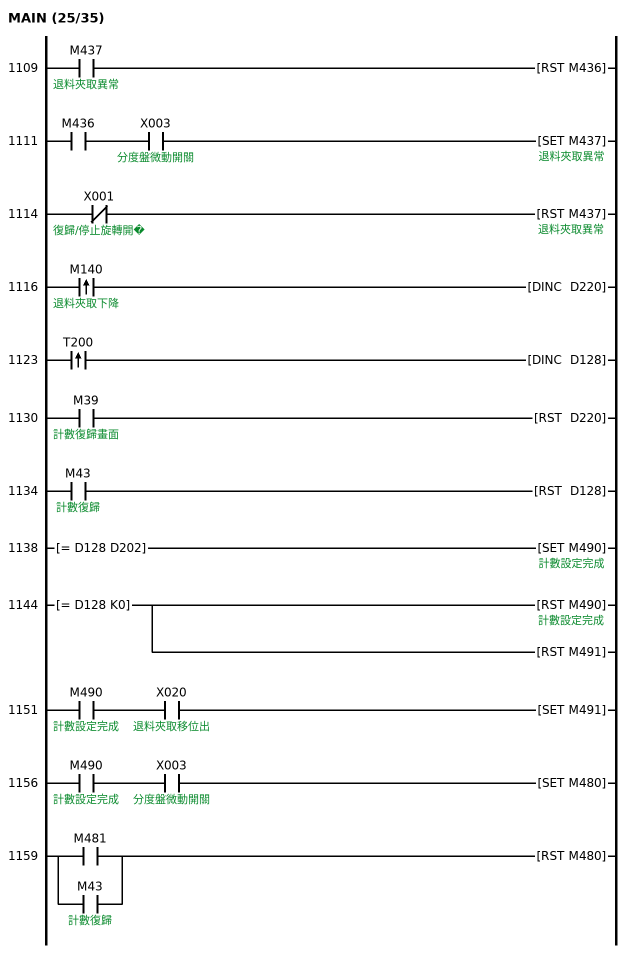
[picture p24: ladder of MAIN, rungs at steps 1109 to 1159]
1109  LD      M437  ; 退料夾取異常
      RST     M436
1111  LD      M436
      AND     X003  ; 分度盤微動開關
      SET     M437  ; 退料夾取異常
1114  LDI     X001  ; 復歸/停止旋轉開�
      RST     M437  ; 退料夾取異常
1116  LDP     M140  ; 退料夾取下降
      DINC    D220
1123  LDP     T200
      DINC    D128
1130  LD      M39  ; 計數復歸畫面
      RST     D220
1134  LD      M43  ; 計數復歸
      RST     D128
1138  LD=     D128 D202
      SET     M490  ; 計數設定完成
1144  LD=     D128 K0
      RST     M490  ; 計數設定完成
      RST     M491
1151  LD      M490  ; 計數設定完成
      AND     X020  ; 退料夾取移位出
      SET     M491
1156  LD      M490  ; 計數設定完成
      AND     X003  ; 分度盤微動開關
      SET     M480
1159  LD      M481
      OR      M43  ; 計數復歸
      RST     M480
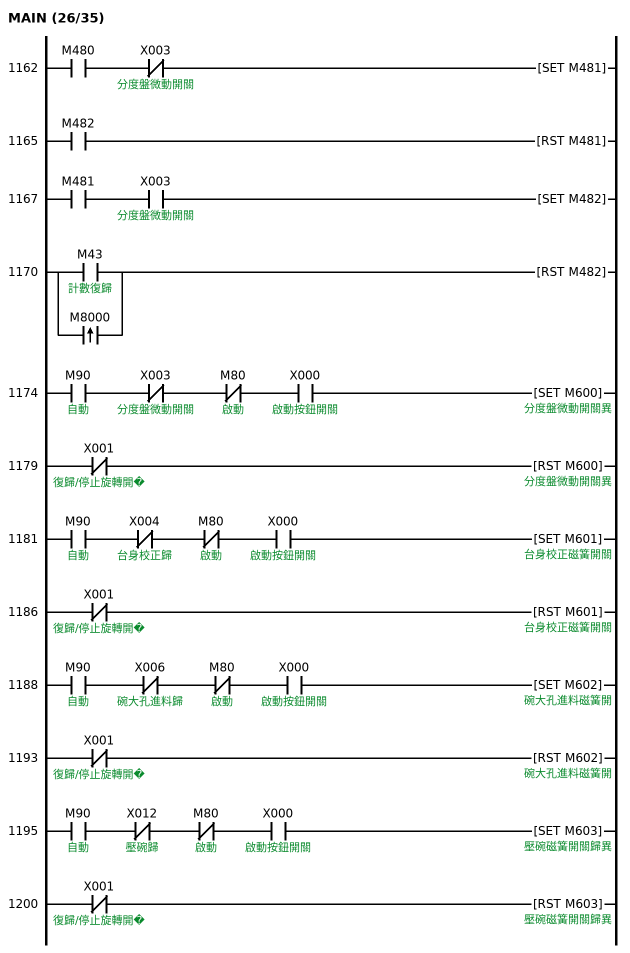
1162  LD      M480
      ANI     X003  ; 分度盤微動開關
      SET     M481
1165  LD      M482
      RST     M481
1167  LD      M481
      AND     X003  ; 分度盤微動開關
      SET     M482
1170  LD      M43  ; 計數復歸
      ORP     M8000
      RST     M482
1174  LD      M90  ; 自動
      ANI     X003  ; 分度盤微動開關
      ANI     M80  ; 啟動
      AND     X000  ; 啟動按鈕開關
      SET     M600  ; 分度盤微動開關異
1179  LDI     X001  ; 復歸/停止旋轉開�
      RST     M600  ; 分度盤微動開關異
1181  LD      M90  ; 自動
      ANI     X004  ; 台身校正歸
      ANI     M80  ; 啟動
      AND     X000  ; 啟動按鈕開關
      SET     M601  ; 台身校正磁簧開關
1186  LDI     X001  ; 復歸/停止旋轉開�
      RST     M601  ; 台身校正磁簧開關
1188  LD      M90  ; 自動
      ANI     X006  ; 碗大孔進料歸
      ANI     M80  ; 啟動
      AND     X000  ; 啟動按鈕開關
      SET     M602  ; 碗大孔進料磁簧開
1193  LDI     X001  ; 復歸/停止旋轉開�
      RST     M602  ; 碗大孔進料磁簧開
1195  LD      M90  ; 自動
      ANI     X012  ; 壓碗歸
      ANI     M80  ; 啟動
      AND     X000  ; 啟動按鈕開關
      SET     M603  ; 壓碗磁簧開關歸異
1200  LDI     X001  ; 復歸/停止旋轉開�
      RST     M603  ; 壓碗磁簧開關歸異
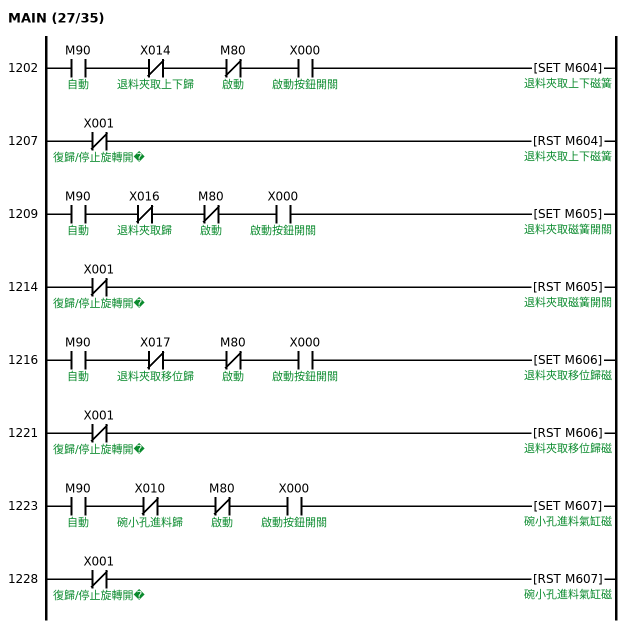
1202  LD      M90  ; 自動
      ANI     X014  ; 退料夾取上下歸
      ANI     M80  ; 啟動
      AND     X000  ; 啟動按鈕開關
      SET     M604  ; 退料夾取上下磁簧
1207  LDI     X001  ; 復歸/停止旋轉開�
      RST     M604  ; 退料夾取上下磁簧
1209  LD      M90  ; 自動
      ANI     X016  ; 退料夾取歸
      ANI     M80  ; 啟動
      AND     X000  ; 啟動按鈕開關
      SET     M605  ; 退料夾取磁簧開關
1214  LDI     X001  ; 復歸/停止旋轉開�
      RST     M605  ; 退料夾取磁簧開關
1216  LD      M90  ; 自動
      ANI     X017  ; 退料夾取移位歸
      ANI     M80  ; 啟動
      AND     X000  ; 啟動按鈕開關
      SET     M606  ; 退料夾取移位歸磁
1221  LDI     X001  ; 復歸/停止旋轉開�
      RST     M606  ; 退料夾取移位歸磁
1223  LD      M90  ; 自動
      ANI     X010  ; 碗小孔進料歸
      ANI     M80  ; 啟動
      AND     X000  ; 啟動按鈕開關
      SET     M607  ; 碗小孔進料氣缸磁
1228  LDI     X001  ; 復歸/停止旋轉開�
      RST     M607  ; 碗小孔進料氣缸磁
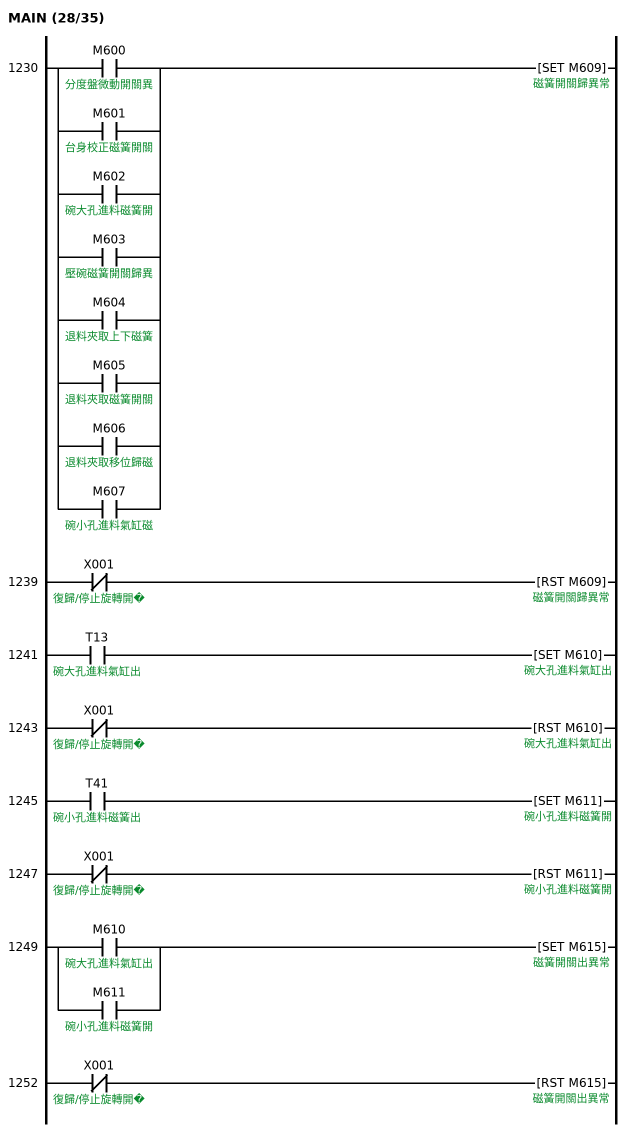
1230  LD      M600  ; 分度盤微動開關異
      OR      M601  ; 台身校正磁簧開關
      OR      M602  ; 碗大孔進料磁簧開
      OR      M603  ; 壓碗磁簧開關歸異
      OR      M604  ; 退料夾取上下磁簧
      OR      M605  ; 退料夾取磁簧開關
      OR      M606  ; 退料夾取移位歸磁
      OR      M607  ; 碗小孔進料氣缸磁
      SET     M609  ; 磁簧開關歸異常
1239  LDI     X001  ; 復歸/停止旋轉開�
      RST     M609  ; 磁簧開關歸異常
1241  LD      T13  ; 碗大孔進料氣缸出
      SET     M610  ; 碗大孔進料氣缸出
1243  LDI     X001  ; 復歸/停止旋轉開�
      RST     M610  ; 碗大孔進料氣缸出
1245  LD      T41  ; 碗小孔進料磁簧出
      SET     M611  ; 碗小孔進料磁簧開
1247  LDI     X001  ; 復歸/停止旋轉開�
      RST     M611  ; 碗小孔進料磁簧開
1249  LD      M610  ; 碗大孔進料氣缸出
      OR      M611  ; 碗小孔進料磁簧開
      SET     M615  ; 磁簧開關出異常
1252  LDI     X001  ; 復歸/停止旋轉開�
      RST     M615  ; 磁簧開關出異常
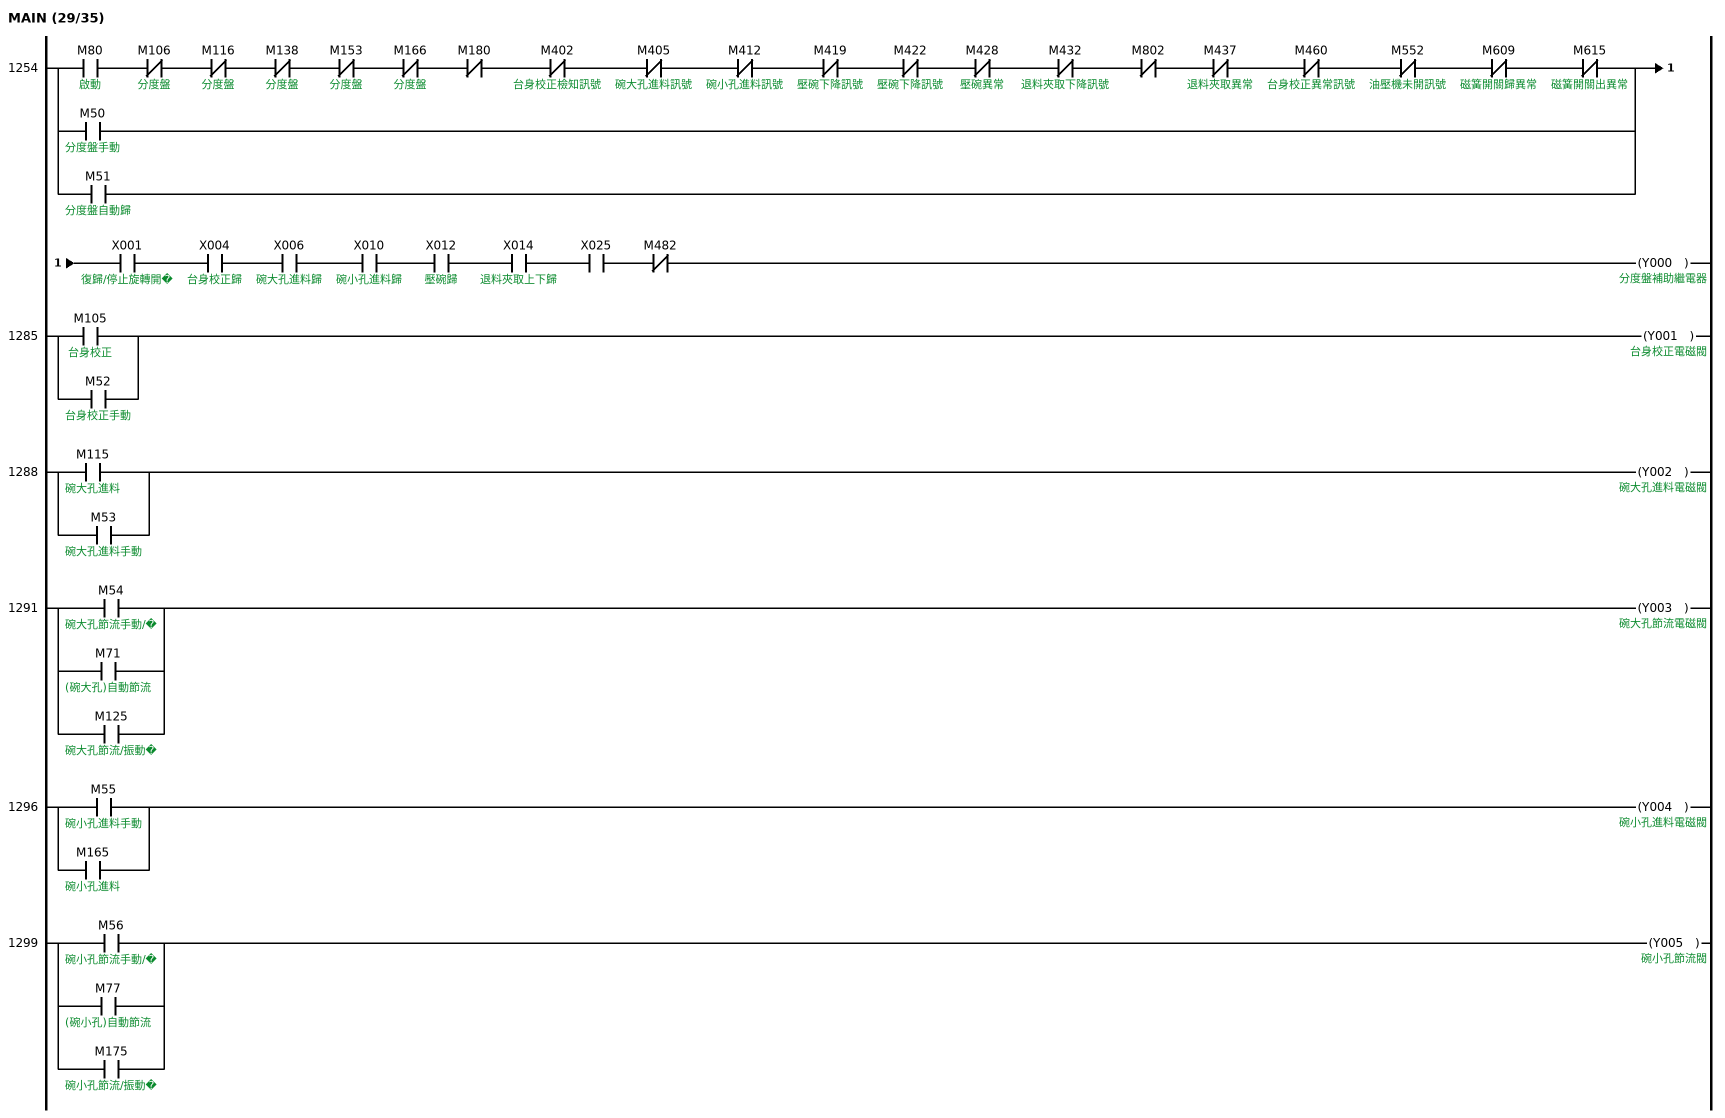
1254  LD      M80  ; 啟動
      ANI     M106  ; 分度盤
      ANI     M116  ; 分度盤
      ANI     M138  ; 分度盤
      ANI     M153  ; 分度盤
      ANI     M166  ; 分度盤
      ANI     M180
      ANI     M402  ; 台身校正檢知訊號
      ANI     M405  ; 碗大孔進料訊號
      ANI     M412  ; 碗小孔進料訊號
      ANI     M419  ; 壓碗下降訊號
      ANI     M422  ; 壓碗下降訊號
      ANI     M428  ; 壓碗異常
      ANI     M432  ; 退料夾取下降訊號
      ANI     M802
      ANI     M437  ; 退料夾取異常
      ANI     M460  ; 台身校正異常訊號
      ANI     M552  ; 油壓機未開訊號
      ANI     M609  ; 磁簧開關歸異常
      ANI     M615  ; 磁簧開關出異常
      OR      M50  ; 分度盤手動
      OR      M51  ; 分度盤自動歸
      AND     X001  ; 復歸/停止旋轉開�
      AND     X004  ; 台身校正歸
      AND     X006  ; 碗大孔進料歸
      AND     X010  ; 碗小孔進料歸
      AND     X012  ; 壓碗歸
      AND     X014  ; 退料夾取上下歸
      AND     X025
      ANI     M482
      OUT     Y000  ; 分度盤補助繼電器
1285  LD      M105  ; 台身校正
      OR      M52  ; 台身校正手動
      OUT     Y001  ; 台身校正電磁閥
1288  LD      M115  ; 碗大孔進料
      OR      M53  ; 碗大孔進料手動
      OUT     Y002  ; 碗大孔進料電磁閥
1291  LD      M54  ; 碗大孔節流手動/�
      OR      M71  ; (碗大孔)自動節流
      OR      M125  ; 碗大孔節流/振動�
      OUT     Y003  ; 碗大孔節流電磁閥
1296  LD      M55  ; 碗小孔進料手動
      OR      M165  ; 碗小孔進料
      OUT     Y004  ; 碗小孔進料電磁閥
1299  LD      M56  ; 碗小孔節流手動/�
      OR      M77  ; (碗小孔)自動節流
      OR      M175  ; 碗小孔節流/振動�
      OUT     Y005  ; 碗小孔節流閥
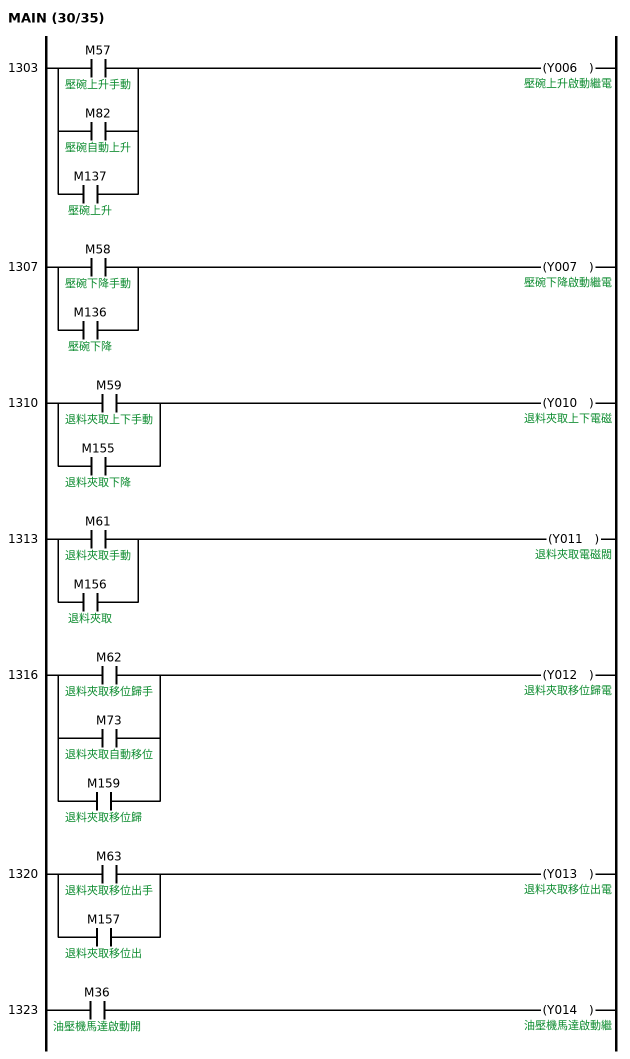
1303  LD      M57  ; 壓碗上升手動
      OR      M82  ; 壓碗自動上升
      OR      M137  ; 壓碗上升
      OUT     Y006  ; 壓碗上升啟動繼電
1307  LD      M58  ; 壓碗下降手動
      OR      M136  ; 壓碗下降
      OUT     Y007  ; 壓碗下降啟動繼電
1310  LD      M59  ; 退料夾取上下手動
      OR      M155  ; 退料夾取下降
      OUT     Y010  ; 退料夾取上下電磁
1313  LD      M61  ; 退料夾取手動
      OR      M156  ; 退料夾取
      OUT     Y011  ; 退料夾取電磁閥
1316  LD      M62  ; 退料夾取移位歸手
      OR      M73  ; 退料夾取自動移位
      OR      M159  ; 退料夾取移位歸
      OUT     Y012  ; 退料夾取移位歸電
1320  LD      M63  ; 退料夾取移位出手
      OR      M157  ; 退料夾取移位出
      OUT     Y013  ; 退料夾取移位出電
1323  LD      M36  ; 油壓機馬達啟動開
      OUT     Y014  ; 油壓機馬達啟動繼
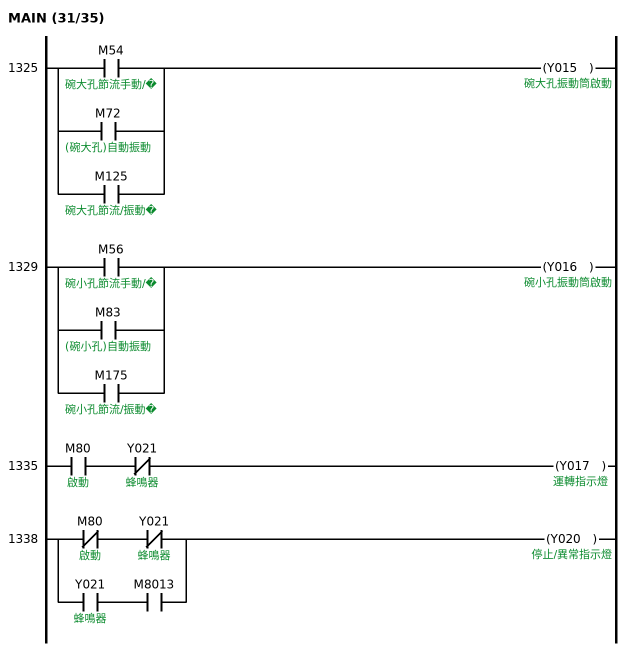
1325  LD      M54  ; 碗大孔節流手動/�
      OR      M72  ; (碗大孔)自動振動
      OR      M125  ; 碗大孔節流/振動�
      OUT     Y015  ; 碗大孔振動筒啟動
1329  LD      M56  ; 碗小孔節流手動/�
      OR      M83  ; (碗小孔)自動振動
      OR      M175  ; 碗小孔節流/振動�
      OUT     Y016  ; 碗小孔振動筒啟動
1335  LD      M80  ; 啟動
      ANI     Y021  ; 蜂鳴器
      OUT     Y017  ; 運轉指示燈
1338  LDI     M80  ; 啟動
      ANI     Y021  ; 蜂鳴器
      LD      Y021  ; 蜂鳴器
      AND     M8013
      ORB
      OUT     Y020  ; 停止/異常指示燈
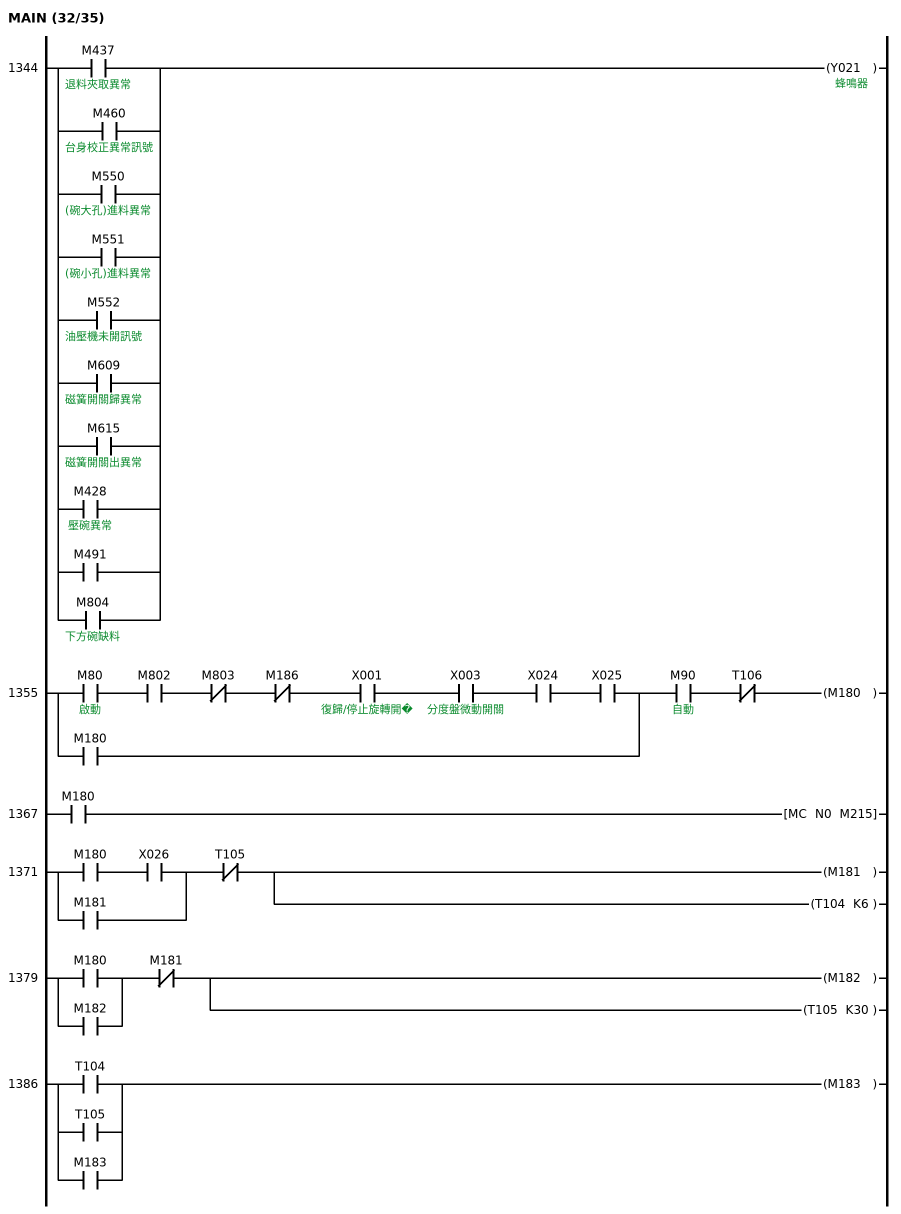
1344  LD      M437  ; 退料夾取異常
      OR      M460  ; 台身校正異常訊號
      OR      M550  ; (碗大孔)進料異常
      OR      M551  ; (碗小孔)進料異常
      OR      M552  ; 油壓機未開訊號
      OR      M609  ; 磁簧開關歸異常
      OR      M615  ; 磁簧開關出異常
      OR      M428  ; 壓碗異常
      OR      M491
      OR      M804  ; 下方碗缺料
      OUT     Y021  ; 蜂鳴器
1355  LD      M80  ; 啟動
      AND     M802
      ANI     M803
      ANI     M186
      AND     X001  ; 復歸/停止旋轉開�
      AND     X003  ; 分度盤微動開關
      AND     X024
      AND     X025
      OR      M180
      AND     M90  ; 自動
      ANI     T106
      OUT     M180
1367  LD      M180
      MC      N0 M215
1371  LD      M180
      AND     X026
      OR      M181
      ANI     T105
      OUT     M181
      OUT     T104 K6
1379  LD      M180
      OR      M182
      ANI     M181
      OUT     M182
      OUT     T105 K30
1386  LD      T104
      OR      T105
      OR      M183
      OUT     M183
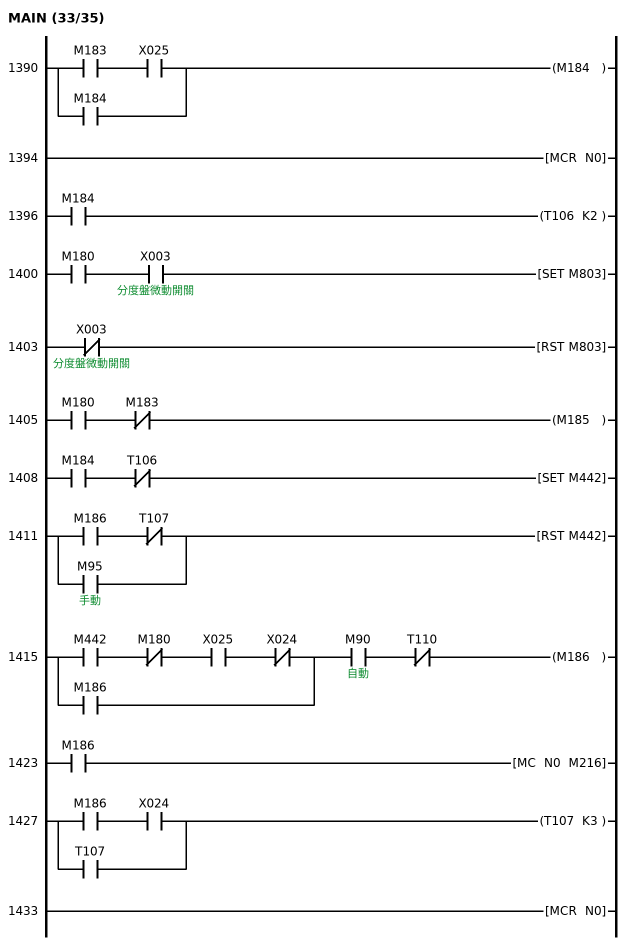
1390  LD      M183
      AND     X025
      OR      M184
      OUT     M184
1394  MCR     N0
1396  LD      M184
      OUT     T106 K2
1400  LD      M180
      AND     X003  ; 分度盤微動開關
      SET     M803
1403  LDI     X003  ; 分度盤微動開關
      RST     M803
1405  LD      M180
      ANI     M183
      OUT     M185
1408  LD      M184
      ANI     T106
      SET     M442
1411  LD      M186
      ANI     T107
      OR      M95  ; 手動
      RST     M442
1415  LD      M442
      ANI     M180
      AND     X025
      ANI     X024
      OR      M186
      AND     M90  ; 自動
      ANI     T110
      OUT     M186
1423  LD      M186
      MC      N0 M216
1427  LD      M186
      AND     X024
      OR      T107
      OUT     T107 K3
1433  MCR     N0
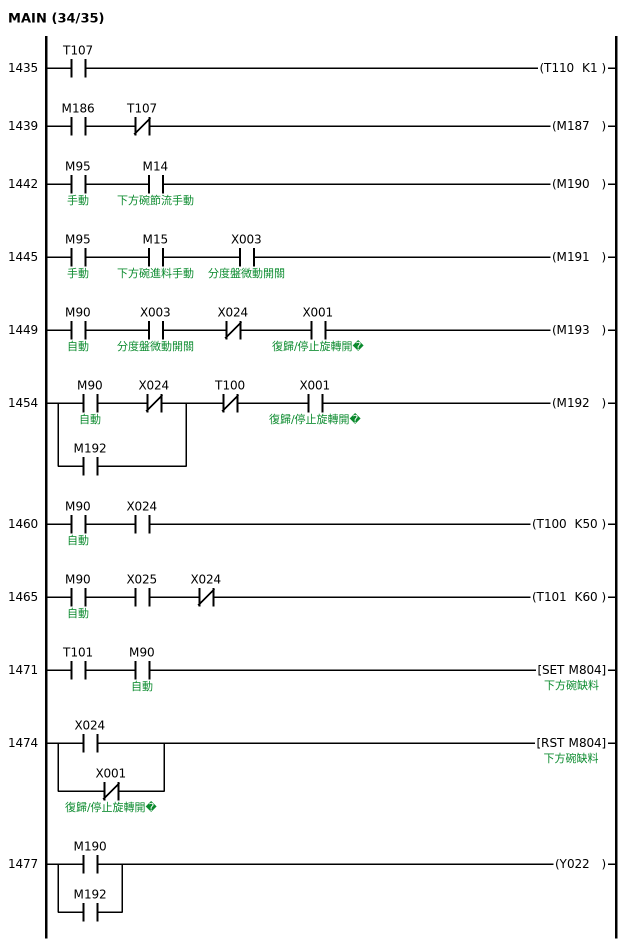
1435  LD      T107
      OUT     T110 K1
1439  LD      M186
      ANI     T107
      OUT     M187
1442  LD      M95  ; 手動
      AND     M14  ; 下方碗節流手動
      OUT     M190
1445  LD      M95  ; 手動
      AND     M15  ; 下方碗進料手動
      AND     X003  ; 分度盤微動開關
      OUT     M191
1449  LD      M90  ; 自動
      AND     X003  ; 分度盤微動開關
      ANI     X024
      AND     X001  ; 復歸/停止旋轉開�
      OUT     M193
1454  LD      M90  ; 自動
      ANI     X024
      OR      M192
      ANI     T100
      AND     X001  ; 復歸/停止旋轉開�
      OUT     M192
1460  LD      M90  ; 自動
      AND     X024
      OUT     T100 K50
1465  LD      M90  ; 自動
      AND     X025
      ANI     X024
      OUT     T101 K60
1471  LD      T101
      AND     M90  ; 自動
      SET     M804  ; 下方碗缺料
1474  LD      X024
      ORI     X001  ; 復歸/停止旋轉開�
      RST     M804  ; 下方碗缺料
1477  LD      M190
      OR      M192
      OUT     Y022
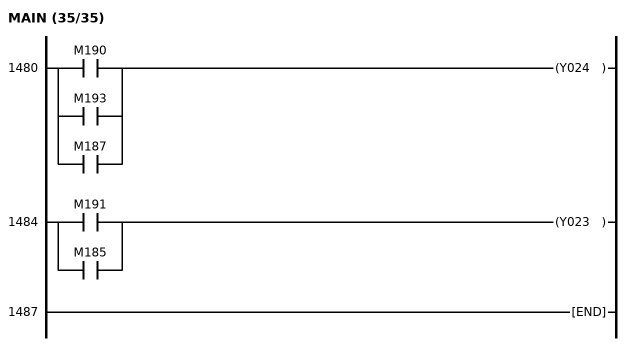
1480  LD      M190
      OR      M193
      OR      M187
      OUT     Y024
1484  LD      M191
      OR      M185
      OUT     Y023
1487  END
END_PROGRAM

// device comments not shown above
M20  ; 碗小孔振動筒
M40  ; 計數復歸畫面
M85  ; 台身進料檢知
M149  ; 退料夾取下降切
M158  ; 退料夾取下降
M176  ; 碗小孔振動筒
M177  ; 碗大孔振動筒
M302  ; 碗小孔節流訊號
M439  ; 退料異常訊號
M612  ; 退料上下磁簧開關
M613  ; 碗小孔進料磁簧開
T0  ; (碗大孔)自動節流
T17  ; 碗大孔缺料訊號
T22  ; 壓碗OK
T33  ; 退料夾取下降
T35  ; 退料夾取下降切
T38  ; 退料夾取下降出異
T44  ; 碗小孔進料異常訊
